// TIA Portal V17 export
// export: Created 2022-07-20T07:02:41.7597394Z, ExportSetting WithDefaults, DisplayName Totally Integrated Automation Portal, DisplayVersion V17, DisplayName TIA Portal Openness, DisplayVersion V17, DisplayName TIA Portal Version Control Interface, DisplayVersion V17, DisplayName SINAMICS Startdrive Advanced, DisplayVersion V17, DisplayName SINAMICS Startdrive G130, G150, S120, S150, SINAMICS MV, S210, DisplayVersion V17, DisplayName SINAMICS Startdrive G110M, G120, G120C, G120D, G120P, G115D, DisplayVersion V17, DisplayName STEP 7 Professional, DisplayVersion V17, DisplayName STEP 7 Safety, DisplayVersion V17, DisplayName WinCC Advanced, DisplayVersion V17
ORGANIZATION_BLOCK "Main"   // OB1, FBD, ProgramCycle
TITLE = "Main Program Sweep (Cycle)"
{ S7_Optimized_Access := 'TRUE' }
VERSION : 0.1
// stored: AutoNumber true, IsIECCheckEnabled false, SetENOAutomatically false
   VAR_INPUT
      Initial_Call : Bool;   // Initial call of this OB
      Remanence : Bool;   // =True, if remanent data are available
   END_VAR
BEGIN

REGION Network 1: Call CTRL_HSC_EXT for HSC1
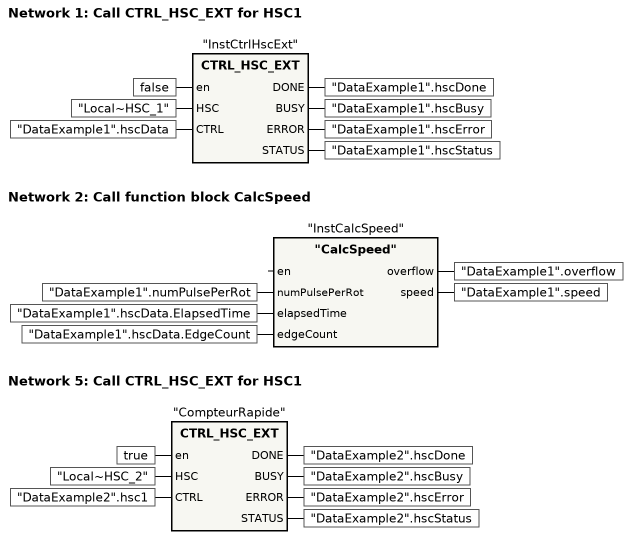
   IF false THEN
       "InstCtrlHscExt"(HSC := "Local~HSC_1",   // CTRL_HSC_EXT
                        CTRL := "DataExample1".hscData,
                        DONE => "DataExample1".hscDone,
                        BUSY => "DataExample1".hscBusy,
                        ERROR => "DataExample1".hscError,
                        STATUS => "DataExample1".hscStatus);
   END_IF;
END_REGION

REGION Network 2: Call function block CalcSpeed
   "InstCalcSpeed"(numPulsePerRot := "DataExample1".numPulsePerRot,   // "CalcSpeed"
                   elapsedTime := "DataExample1".hscData.ElapsedTime,
                   edgeCount := "DataExample1".hscData.EdgeCount,
                   overflow => "DataExample1".overflow,
                   speed => "DataExample1".speed);
END_REGION

REGION Network 3 (SCL)
   "DataExample1".vitesse := 0.2 * "DataExample1".speed;
END_REGION

REGION Network 5: Call CTRL_HSC_EXT for HSC1
   IF true THEN
       "CompteurRapide"(HSC := "Local~HSC_2",   // CTRL_HSC_EXT
                        CTRL := "DataExample2".hsc1,
                        DONE => "DataExample2".hscDone,
                        BUSY => "DataExample2".hscBusy,
                        ERROR => "DataExample2".hscError,
                        STATUS => "DataExample2".hscStatus);
   END_IF;
END_REGION
END_ORGANIZATION_BLOCK
